Staubli VAL3: onF4Event.pgx

public program onF4Event()
begin
end
